(* IEC 61131-3 sources: stformat/handlers/testdata, 60 files *)

(* ---- dut_pragma.golden.iecst ---- *)
{attribute 'qualified_only'}

TYPE S :
	( // Some comment
		A := 10,
		B := 20,
		C := 30,
		D := 40,
		E := 50,
		F := 60,
		G := 70,
		H := 80,
		I := 90,
		J := 100,
		K := 110,
		L := 120,
		M := 130,
		N := 140,
		P := 150
	);
END_TYPE

(* ---- dut_pragma.in.iecst ---- *)
{attribute 'qualified_only'}

TYPE S :
	(  // Some comment
		A := 10, B := 20, C := 30, D := 40, E := 50, F := 60, G := 70, H := 80, I := 90, J := 100, K := 110, L := 120, M := 130, N := 140, P := 150
	);
END_TYPE

(* ---- type_body.golden.st ---- *)
// The value list of a TYPE.
// A TYPE body is a list of values like a call's argument list, so it breaks at the same limit into the same layout.
// The bracket depth is carried from line to line, and text that is not structure must not feed it.

// A body over the limit breaks one member per line.

TYPE EState :
	(
		A := 0,
		B := 1,
		C := 2,
		D := 3,
		E := 4,
		F := 5,
		G := 6,
		H := 7,
		I := 8,
		J := 9,
		K := 10,
		L := 11,
		M := 12,
		N := 13,
		O := 14,
		P := 15
	);
END_TYPE

// One member cannot be split any further, so the line stays long.

TYPE t :
	(
		A := 1000000000000000000000000000000000000000000000000000000000000000000000000000000000000000000000000000000000
	);
END_TYPE

// A parenthesis inside a comment is text, so it does not open a level.
(* note ( unbalanced *)

TYPE FromComment :
	(
		A := 0,
		B := 1,
		C := 2,
		D := 3,
		E := 4,
		F := 5,
		G := 6,
		H := 7,
		I := 8,
		J := 9,
		K := 10,
		L := 11,
		M := 12,
		N := 13,
		O := 14,
		P := 15
	);
END_TYPE

// Same for an ignored region: the count restarts at stformat:on.

TYPE FromRegion :
	// stformat:off
weird ( unbalanced ( ( (
	// stformat:on
	(
		A := 0,
		B := 1,
		C := 2,
		D := 3,
		E := 4,
		F := 5,
		G := 6,
		H := 7,
		I := 8,
		J := 9,
		K := 10,
		L := 11,
		M := 12,
		N := 13,
		O := 14,
		P := 15
	);
END_TYPE

(* ---- type_body.in.st ---- *)
// The value list of a TYPE.
// A TYPE body is a list of values like a call's argument list, so it breaks at the same limit into the same layout.
// The bracket depth is carried from line to line, and text that is not structure must not feed it.

// A body over the limit breaks one member per line.
TYPE EState :
(A := 0, B := 1, C := 2, D := 3, E := 4, F := 5, G := 6, H := 7, I := 8, J := 9, K := 10, L := 11, M := 12, N := 13, O := 14, P := 15);
END_TYPE

// One member cannot be split any further, so the line stays long.
TYPE t :
(A := 1000000000000000000000000000000000000000000000000000000000000000000000000000000000000000000000000000000000);
END_TYPE

// A parenthesis inside a comment is text, so it does not open a level.
(* note ( unbalanced *)
TYPE FromComment :
(A := 0, B := 1, C := 2, D := 3, E := 4, F := 5, G := 6, H := 7, I := 8, J := 9, K := 10, L := 11, M := 12, N := 13, O := 14, P := 15);
END_TYPE

// Same for an ignored region: the count restarts at stformat:on.
TYPE FromRegion :
// stformat:off
weird ( unbalanced ( ( (
// stformat:on
(A := 0, B := 1, C := 2, D := 3, E := 4, F := 5, G := 6, H := 7, I := 8, J := 9, K := 10, L := 11, M := 12, N := 13, O := 14, P := 15);
END_TYPE

(* ---- types.golden.st ---- *)
TYPE point :
	STRUCT
		x : INT;
		y : INT;
	END_STRUCT

	union32 : UNION
		a : INT;
		b : DWORD;
		c : REAL;
	END_UNION

	matrix : ARRAY[1..3, 1..3] OF REAL;
	point_arr : ARRAY[1..4] OF point;
END_TYPE

(* ---- types.in.st ---- *)
type
point:
struct
x: int;
y: int;
end_struct
union32:
union
a: int;
b: dword;
c: real;
end_union
matrix: array[1..3,1..3] of real;
point_arr: array[1..4] of point;
end_type

(* ---- comments.golden.st ---- *)
PROGRAM p
VAR
	x : INT; // the counter
END_VAR

x := 1; // set x
(* block
comment *)
z := 2;
IF x THEN
	y := x; // branch
END_IF // done
(* note *)
z := 3;
END_PROGRAM

// A comment standing on its own line inside a condition.
// The tokens around it ask for no line break, so a second pass used to glue it to the line above.

PROGRAM p
IF a
// both must be set
AND b THEN
	c := 1;
END_IF
END_PROGRAM

// A trailing comment on a condition that has to wrap moves to the THEN line.

PROGRAM p
IF flagOperationalReady
	AND flagMaintenanceOverride
	AND flagEmergencyStopActive
	AND flagPowerAvailable
	AND flagGateClosed
	AND flagInterlockEngaged
	AND flagSequenceRunning
	AND flagAbortRequested
	AND flagResetPermitted
	AND flagCycleComplete
	AND flagAutoModeSelected
THEN // all flags
	x := TRUE;
END_IF
END_PROGRAM

FUNCTION_BLOCK fb EXTENDS base
// built by the comment test
VAR
	y : INT;
END_VAR

y := 1;
END_FUNCTION_BLOCK

// a type with the comment on the line that opens its body

TYPE states :
	(
		// the state names
		a := 0,
		b := 1
	);
END_TYPE

FUNCTION_BLOCK child PUBLIC EXTENDS base
// inherits from base
VAR
	w : INT;
END_VAR
END_FUNCTION_BLOCK
(*****************)
//////////
///doc comment
// x := 1; commented-out code keeps its case
//   indented text keeps its indentation

(* ---- comments.in.st ---- *)
program p
VAR
x:int; //the counter
END_VAR
x:=1; //set x
(* block
comment *)
z:=2;
if x then
    y:=x; //branch
end_if //done
(* note *) z := 3;
end_program

// A comment standing on its own line inside a condition.
// The tokens around it ask for no line break, so a second pass used to glue it to the line above.
program p
IF a
// both must be set
AND b THEN c := 1; END_IF
end_program

// A trailing comment on a condition that has to wrap moves to the THEN line.
program p
IF flagOperationalReady AND flagMaintenanceOverride AND flagEmergencyStopActive AND flagPowerAvailable AND flagGateClosed AND flagInterlockEngaged AND flagSequenceRunning AND flagAbortRequested AND flagResetPermitted AND flagCycleComplete AND flagAutoModeSelected THEN // all flags
    x := TRUE;
END_IF
end_program

function_block fb extends base
// built by the comment test
var
    y:int;
end_var
y:=1;
end_function_block

// a type with the comment on the line that opens its body
type states :
(
// the state names
a:=0,
b:=1
);
end_type

function_block child public extends base
// inherits from base
var
    w:int;
end_var
end_function_block
(*****************)
//////////
///doc comment
//x := 1; commented-out code keeps its case
//   indented text keeps its indentation

(* ---- constructs.golden.st ---- *)
// Namespaces, configurations, property accessors and SFC, whose openers are
// recognised only where their closing keyword follows.

NAMESPACE Motion

FUNCTION F_A : INT
F_A := 1;
END_FUNCTION

FUNCTION F_B : INT
F_B := 2;
END_FUNCTION
END_NAMESPACE

CONFIGURATION Cell
	VAR_GLOBAL
		bRun : BOOL;
	END_VAR

	RESOURCE Cpu ON PLC
		TASK Fast(INTERVAL := T#10MS, PRIORITY := 1);
		PROGRAM Main WITH Fast : P_Main;
	END_RESOURCE
END_CONFIGURATION

FUNCTION_BLOCK FB_Prop
PROPERTY Value : INT
GET
Value := nValue;
END_GET
SET
nValue := Value;
END_SET
END_PROPERTY
END_FUNCTION_BLOCK

PROGRAM Chart
INITIAL_STEP Idle:
	Reset(N);
END_STEP

STEP Run:
	Drive(N);
END_STEP

TRANSITION FROM Idle TO Run := bStart;
END_TRANSITION
END_PROGRAM

// The same words used as names stay names.

PROGRAM Names
VAR
	Step, Set, Get : INT;
END_VAR

Step := Step + 1;
Set := Get;
fb.Set(1);
IF Step > 3 THEN
	Step := 0;
END_IF
END_PROGRAM

// An opener right after a POU header, with no VAR block between.

PROGRAM Direct
STEP Run:
	DriveTheAxisToPosition(Position := fTargetPositionInMillimetres, Velocity := fVelocityLimit, Acceleration := fAcc);
END_STEP
END_PROGRAM

(* ---- constructs.in.st ---- *)
// Namespaces, configurations, property accessors and SFC, whose openers are
// recognised only where their closing keyword follows.
NAMESPACE Motion
FUNCTION F_A : INT
F_A := 1;
END_FUNCTION
FUNCTION F_B : INT
F_B := 2;
END_FUNCTION
END_NAMESPACE

CONFIGURATION Cell
VAR_GLOBAL bRun : BOOL; END_VAR
RESOURCE Cpu ON PLC
TASK Fast(INTERVAL := T#10MS, PRIORITY := 1);
PROGRAM Main WITH Fast : P_Main;
END_RESOURCE
END_CONFIGURATION

FUNCTION_BLOCK FB_Prop
PROPERTY Value : INT
GET
Value := nValue;
END_GET
SET
nValue := Value;
END_SET
END_PROPERTY
END_FUNCTION_BLOCK

PROGRAM Chart
INITIAL_STEP Idle: Reset(N);
END_STEP
STEP Run: Drive(N);
END_STEP
TRANSITION FROM Idle TO Run := bStart;
END_TRANSITION
END_PROGRAM

// The same words used as names stay names.
PROGRAM Names
VAR Step, Set, Get : INT; END_VAR
Step := Step + 1;
Set := Get;
fb.Set(1);
IF Step > 3 THEN Step := 0; END_IF
END_PROGRAM

// An opener right after a POU header, with no VAR block between.
PROGRAM Direct
STEP Run:
DriveTheAxisToPosition(Position := fTargetPositionInMillimetres, Velocity := fVelocityLimit, Acceleration := fAcc);
END_STEP
END_PROGRAM

(* ---- functions.golden.st ---- *)
FUNCTION max2 : INT
max2 := a;
END_FUNCTION

FUNCTION_BLOCK motor
VAR_INPUT
	cmd : BOOL;
	speed : REAL;
END_VAR

METHOD Execute : BOOL
VAR
	result : BOOL;
END_VAR

result := cmd;
END_METHOD
ACTION do_it
speed := 10.0;
END_ACTION
END_FUNCTION_BLOCK

FUNCTION combine : INT
combine := max2(1, 2);
END_FUNCTION

(* ---- functions.in.st ---- *)
function max2: int
max2:=a;
end_function
function_block motor
var_input
cmd: bool;
speed: real;
end_var
method Execute: bool
var
result: bool;
end_var
result:=cmd;
end_method
action do_it
speed:=10.0;
end_action
end_function_block
function combine: int
combine:=max2(1,2);
end_function

(* ---- headers.golden.st ---- *)
// POU and member headers: modifiers, return types and inheritance lists.

FUNCTION F_Ptr : POINTER TO INT
VAR_INPUT
	a : INT;
END_VAR

F_Ptr := ADR(a);
END_FUNCTION

FUNCTION F_Arr : ARRAY[0..1, 1..2] OF INT
END_FUNCTION

FUNCTION F_Str : STRING(80)
END_FUNCTION

FUNCTION F_Ns : Lib.ST_Data
END_FUNCTION

FUNCTION_BLOCK PUBLIC ABSTRACT FB_X EXTENDS FB_Base IMPLEMENTS I_A, Lib.I_B
VAR
END_VAR

METHOD PUBLIC ABSTRACT M : REFERENCE TO INT
VAR_INPUT
	x : INT;
END_VAR
END_METHOD

METHOD FINAL PROTECTED M2 : BOOL
END_METHOD

PROPERTY PUBLIC P : POINTER TO FB_X
END_PROPERTY
END_FUNCTION_BLOCK

INTERFACE I_A EXTENDS I_Base, I_Other
METHOD M : BOOL
END_METHOD
END_INTERFACE

FUNCTION_BLOCK FB_G
VAR_GENERIC CONSTANT
	N : UDINT := 10;
END_VAR
END_FUNCTION_BLOCK

(* ---- headers.in.st ---- *)
// POU and member headers: modifiers, return types and inheritance lists.
FUNCTION F_Ptr : POINTER TO INT
VAR_INPUT a:INT; END_VAR
F_Ptr := ADR(a);
END_FUNCTION

function F_Arr : array[0..1, 1..2] of int
END_FUNCTION

FUNCTION F_Str : STRING(80)
END_FUNCTION

FUNCTION F_Ns : Lib.ST_Data
END_FUNCTION

function_block public abstract FB_X extends FB_Base implements I_A, Lib.I_B
VAR END_VAR

METHOD public abstract M : reference to INT
VAR_INPUT x : INT; END_VAR
END_METHOD

METHOD final protected M2 : BOOL
END_METHOD

PROPERTY PUBLIC P : POINTER TO FB_X
END_PROPERTY
END_FUNCTION_BLOCK

INTERFACE I_A EXTENDS I_Base, I_Other
METHOD M : BOOL
END_METHOD
END_INTERFACE

FUNCTION_BLOCK FB_G
VAR_GENERIC CONSTANT
N : UDINT := 10;
END_VAR
END_FUNCTION_BLOCK

(* ---- oostuff.golden.st ---- *)
CLASS my_class EXTENDS base
VAR
	x : INT;
END_VAR

METHOD PUBLIC compute : INT
compute := x * 2;
END_METHOD
METHOD PROTECTED helper : INT
helper := THIS.x + SUPER.get();
END_METHOD
METHOD ABSTRACT enforce
END_METHOD
METHOD FINAL lockit
register := 1;
END_METHOD
PROPERTY PRIVATE value : INT
END_PROPERTY
END_CLASS

INTERFACE my_interface
METHOD PUBLIC cycle : INT
END_METHOD
METHOD PROTECTED semi : INT
END_METHOD
END_INTERFACE

FUNCTION_BLOCK axis IMPLEMENTS i_motion
VAR
	pos : INT;
END_VAR

METHOD PUBLIC move : INT
move := pos;
END_METHOD
END_FUNCTION_BLOCK

(* ---- oostuff.in.st ---- *)
class my_class extends base
var
x: int;
end_var
method public compute: int
compute:=x*2;
end_method
method protected helper: int
helper:=this.x + super.get();
end_method
method abstract enforce
end_method
method final lockit
register:=1;
end_method
property private value: int
end_property
end_class
interface my_interface
method public cycle: int
end_method
method protected semi: int
end_method
end_interface
function_block axis implements i_motion
var
pos: int;
end_var
method public move: int
move:=pos;
end_method
end_function_block

(* ---- addresses.golden.st ---- *)
PROGRAM p
VAR
	inBit : BOOL AT %i*;
	outBit : BOOL AT %q*;
	inByte : BYTE AT %ib3;
	inWord : WORD AT %IW50;
	outBit2 : BOOL AT %Q0.0;
	memWord : WORD AT %MW100;
	memByte : BYTE AT %MB128;
	memDword : DWORD AT %MD1000;
	memBit : BOOL AT %M0.3;
END_VAR
END_PROGRAM

(* ---- addresses.in.st ---- *)
program p
var
inBit: bool at %i*;
outBit: bool at %q*;
inByte: byte at %ib3;
inWord: word at %IW50;
outBit2: bool at %Q0.0;
memWord: word at %MW100;
memByte: byte at %MB128;
memDword: dword at %MD1000;
memBit: bool at %M0.3;
end_var
end_program

(* ---- bindings.golden.st ---- *)
PROGRAM p
VAR
	setOut : BOOL;
	resetOut : BOOL;
	bitUp : BOOL;
	bitDown : BOOL;
	pSrc : POINTER TO INT;
	pDst : POINTER TO INT;
	pref : REFERENCE TO INT;
	refTo : REF_TO INT;
	pInst : POINTER TO INT;
	pTmp : POINTER TO INT;
	valid : BOOL;
	rAxis : REAL;
	fb : fb_axis;
END_VAR

setOut s= bitUp;
resetOut r= bitDown;
pDst ref= pSrc;
pDst^ := 1;
pref^ := 2;
refTo := fb;
pInst := __NEW(pTmp);
__DELETE(pInst);
valid := __ISVALIDREF(pref);
rAxis := fb.mv(velocity := 100.0);
END_PROGRAM

(* ---- bindings.in.st ---- *)
program p
var
setOut: bool;
resetOut: bool;
bitUp: bool;
bitDown: bool;
pSrc: pointer to int;
pDst: pointer to int;
pref: reference to int;
refTo: ref_to int;
pInst: pointer to int;
pTmp: pointer to int;
valid: bool;
rAxis: real;
fb: fb_axis;
end_var
setOut s= bitUp;
resetOut r= bitDown;
pDst ref= pSrc;
pDst^ := 1;
pref^ := 2;
refTo := fb;
pInst := __NEW(pTmp);
__DELETE(pInst);
valid := __ISVALIDREF(pref);
rAxis := fb.mv(velocity := 100.0);
end_program

(* ---- bom.golden.st ---- *)
// A UTF-8 byte order mark is kept.

PROGRAM bom
x := 1;
END_PROGRAM

(* ---- bom.in.st ---- *)
// A UTF-8 byte order mark is kept.
PROGRAM bom
x:=1;
END_PROGRAM

(* ---- control_flow.golden.st ---- *)
PROGRAM p
VAR
	x : BOOL;
	y : INT;
END_VAR

IF x THEN
	x := TRUE;
ELSIF y > 3 THEN
	y := y + 1;
ELSE
	y := 0;
END_IF

FOR i := 1 TO 10 BY 2 DO
	IF y > 5 THEN
		EXIT;
	END_IF

	i := i + 1;
END_FOR

WHILE x DO
	x := FALSE;
END_WHILE

REPEAT
	y := y - 1;
UNTIL y = 0
END_REPEAT

CASE i OF
	1:
		x := TRUE;

	2, 3:
		y := 5;

	4:
		IF x THEN
			x := TRUE;
		END_IF

	5:
		y := 7;
	ELSE
		y := 0;
END_CASE
END_PROGRAM

(* ---- control_flow.in.st ---- *)
program p
var
x: bool;
y: int;
end_var
if x then
x:=true;
elsif y>3 then
y:=y+1;
else
y:=0;
end_if
for i:=1 to 10 by 2 do
if y>5 then
exit;
end_if
i:=i+1;
end_for
while x do
x:=false;
end_while
repeat
y:=y-1;
until y=0 end_repeat
case i of
1: x:=true;
2,3: y:=5;
4:
if x then
x:=true;
end_if 5: y:=7;
else y:=0;
end_case
end_program

(* ---- directives.golden.st ---- *)
PROGRAM Sections
VAR
	a : INT;
END_VAR

// stformat:off
VAR
	ugly    :   INT;
END_VAR
// stformat:on

a := 1; // stformat:off
   b   :=   2;
// stformat:on

(* stformat:off *)
	untouched   :=   1;
(* stformat:on *)

// STFORMAT: OFF
   another    :=   2;
// stformat : on

// stformat:ignore is only a directive in the leading comment block, so here it
// is an ordinary comment.
b := 4; // stformat:ignore
c := 5;

IF a > 0 THEN
	aLongFunctionName(
		firstArgument := aValueWithALongName,
		secondArgument := anotherValueWithALongName,
		thirdArgument := yetAnotherValue
	); // an explanation of the call
END_IF
END_PROGRAM

(* ---- directives.in.st ---- *)
PROGRAM Sections
VAR
	a : INT;
END_VAR

// stformat:off
VAR
	ugly    :   INT;
END_VAR
// stformat:on

a := 1; // stformat:off
   b   :=   2;
// stformat:on

(* stformat:off *)
	untouched   :=   1;
(* stformat:on *)

// STFORMAT: OFF
   another    :=   2;
// stformat : on

// stformat:ignore is only a directive in the leading comment block, so here it
// is an ordinary comment.
b := 4; // stformat:ignore
c := 5;

IF a > 0 THEN
	aLongFunctionName(firstArgument := aValueWithALongName, secondArgument := anotherValueWithALongName, thirdArgument := yetAnotherValue); // an explanation of the call
END_IF
END_PROGRAM

(* ---- expressions.golden.st ---- *)
PROGRAM p
x := (a AND_THEN b) OR_ELSE (c XOR d);
y := NOT(a AND b);
z := a MOD 7;
w := x ** 2;
q := (len > 0) AND (val <> 0);
cmp := (p^ <> meta.q) OR (r <= 5.0);
END_PROGRAM

(* ---- expressions.in.st ---- *)
program p
x := (a and_then b) or_else (c xor d);
y := not (a and b);
z := a mod 7;
w := x ** 2;
q := (len > 0) and (val <> 0);
cmp := (p^ <> meta.q) or (r <= 5.0);
end_program

(* ---- ignore.golden.st ---- *)
// stformat:ignore
PROGRAM Untouched
    x:=1;
IF   x>0   THEN
	y:=2;
END_IF
END_PROGRAM

(* ---- ignore.in.st ---- *)
// stformat:ignore
PROGRAM Untouched
    x:=1;
IF   x>0   THEN
	y:=2;
END_IF
END_PROGRAM

(* ---- illegal.golden.st ---- *)
// Characters that are not ST are kept, with the spacing they had.

PROGRAM illegal
x := y ? 1;
x := y?1;
a := b&c;
Drehzahl_Ä := Größe;
END_PROGRAM

(* ---- illegal.in.st ---- *)
// Characters that are not ST are kept, with the spacing they had.
PROGRAM illegal
x:=y ? 1;
x:=y?1;
a:=b&c;
Drehzahl_Ä:=Größe;
END_PROGRAM

(* ---- line_breaks.golden.st ---- *)
// Line breaks in the source are kept where they mean something, and dropped everywhere else.
// A break after an opening bracket, around a comma or before a closing bracket keeps that list
// broken open, one item per line. A break before or after an operator keeps that chain broken.

// The list is broken in the source, so it stays broken although it fits.

PROGRAM keptList
result := Combine(
	first := 1,
	second := 2
);
END_PROGRAM

// A break after a comma is enough.

PROGRAM keptListAtComma
result := Combine(
	first := 1,
	second := 2
);
END_PROGRAM

// The chain is broken in the source, so every operator of it starts a line.

PROGRAM keptChain
total := a
	+ b
	+ c;
END_PROGRAM

// The break can also come before the operator.

PROGRAM keptChainBefore
ready := sensorOne
	AND sensorTwo
	AND sensorThree;
END_PROGRAM

// A broken condition is laid out in full.

PROGRAM keptCondition
IF a
	OR b
THEN
	x := 1;
END_IF
END_PROGRAM

// Breaks anywhere else are dropped: after the assignment, between a name and its bracket,
// and inside a list that is not broken at one of its own break points.

PROGRAM dropped
x := 5;
y := F(first := 1, second := 2);
z := Compute(a := 1);
END_PROGRAM

// A broken enum stays broken; one written on a line stays on it.

TYPE E_Broken :
	(
		Idle := 0,
		Running := 1
	);
END_TYPE

TYPE E_Inline :
	(
		Idle := 0,
		Running := 1
	);
END_TYPE

(* ---- line_breaks.in.st ---- *)
// Line breaks in the source are kept where they mean something, and dropped everywhere else.
// A break after an opening bracket, around a comma or before a closing bracket keeps that list
// broken open, one item per line. A break before or after an operator keeps that chain broken.

// The list is broken in the source, so it stays broken although it fits.
PROGRAM keptList
result := Combine(
    first := 1, second := 2);
END_PROGRAM

// A break after a comma is enough.
PROGRAM keptListAtComma
result := Combine(first := 1,
    second := 2);
END_PROGRAM

// The chain is broken in the source, so every operator of it starts a line.
PROGRAM keptChain
total := a +
    b + c;
END_PROGRAM

// The break can also come before the operator.
PROGRAM keptChainBefore
ready := sensorOne
    AND sensorTwo AND sensorThree;
END_PROGRAM

// A broken condition is laid out in full.
PROGRAM keptCondition
IF a
    OR b THEN
    x := 1;
END_IF
END_PROGRAM

// Breaks anywhere else are dropped: after the assignment, between a name and its bracket,
// and inside a list that is not broken at one of its own break points.
PROGRAM dropped
x :=
    5;
y := F(first :=
    1, second := 2);
z := Compute
    (a := 1);
END_PROGRAM

// A broken enum stays broken; one written on a line stays on it.
TYPE E_Broken :
(
    Idle := 0,
    Running := 1
);
END_TYPE

TYPE E_Inline :
(Idle := 0, Running := 1);
END_TYPE

(* ---- literal_spans.golden.st ---- *)
// A literal's text must stop where the literal stops.
// A duration that runs into the code after it swallows that code, and a string spanning lines gets a line break put inside quoted text.

// The duration payload stops at the unit. "T#0MS THEN" read as one token loses the rest of the line.

PROGRAM durationThen
IF i_risingDebounceTime <> T#0MS THEN
	m_risingDebounceTimer(IN := m_state, PT := i_risingDebounceTime);
	IF m_risingDebounceTimer.Q THEN
		updateDebounceState := TRUE;
	END_IF
END_IF

IF x > T#0S THEN
	y := z;
END_IF
END_PROGRAM

// The same, with the assignment and the call after the literal.

PROGRAM durationThenMore
IF t^.p > T#0MS THEN
	p := t^.p;
END_IF

IF r <> T#0S THEN
	a := b := r;
END_IF

IF timer.Q OR d = T#0MS THEN
	c := s;
END_IF

IF ts.e > T#0MS THEN
	x := ts.a + ts.b + ts.c;
END_IF

IF ts.e > T#0MS THEN
	calc(IN := TRUE);
END_IF
END_PROGRAM

// A duration with spaced components is one literal, so the blank inside it is kept.

PROGRAM durationSpaced
a := T#1h 30m 20s;
b := LT#2d 12h;
c := TIME#500ms;
d := T#0MS;
END_PROGRAM

// A string spanning lines is one token, so the comma on the next line is content.

PROGRAM stringSpanningLines
log(
	a := 1,
	fmt := 'first,
second',
	b := 2
);
END_PROGRAM

(* ---- literal_spans.in.st ---- *)
// A literal's text must stop where the literal stops.
// A duration that runs into the code after it swallows that code, and a string spanning lines gets a line break put inside quoted text.

// The duration payload stops at the unit. "T#0MS THEN" read as one token loses the rest of the line.
PROGRAM durationThen
IF i_risingDebounceTime <> T#0MS THEN m_risingDebounceTimer(IN := m_state, PT := i_risingDebounceTime);
IF m_risingDebounceTimer.Q THEN updateDebounceState := TRUE; END_IF END_IF
IF x > T#0S THEN y := z;
END_IF
END_PROGRAM

// The same, with the assignment and the call after the literal.
PROGRAM durationThenMore
IF t^.p > T#0MS THEN p := t^.p; END_IF
IF r <> T#0S THEN a := b := r; END_IF
IF timer.Q OR d = T#0MS  THEN c := s; END_IF
IF ts.e > T#0MS THEN x := ts.a + ts.b + ts.c; END_IF
IF ts.e > T#0MS THEN calc(IN := TRUE);
END_IF
END_PROGRAM

// A duration with spaced components is one literal, so the blank inside it is kept.
PROGRAM durationSpaced
a:=T#1h 30m 20s;
b:=LT#2d 12h;
c:=TIME#500ms;
d:=T#0MS;
END_PROGRAM

// A string spanning lines is one token, so the comma on the next line is content.
PROGRAM stringSpanningLines
log(
a := 1,
fmt := 'first,
second',
b := 2
);
END_PROGRAM

(* ---- literals.golden.st ---- *)
PROGRAM p
VAR
	hexVal : DWORD := 16#FF;
	binVal : BYTE := 2#1011;
	octVal : BYTE := 8#77;
	mask : DWORD := 16#FFFFFFFF;
	intTyped : DINT := DINT#-32768;
	wordTyped : WORD := WORD#16#ABCD;
	realTyped : REAL := REAL#1.5;
	boolTyped : BOOL := BOOL#TRUE;
	expVal : REAL := 1.5e3;
	negExp : LREAL := 1.5E-3;
	dur1 : TIME := T#1H 30M 20S 500MS;
	dur2 : TIME := TIME#5S;
	dur3 : LTIME := LTIME#100NS;
	todVal : TOD := TOD#12:30:45.5;
	dateVal : DATE := DATE#2024-06-15;
	dtVal : DT := DT#2024-06-15-12:30:45;
	ldtVal : LDT := LDT#2024-06-15-12:30:45.123;
	str1 : STRING := 'plain';
	str2 : WSTRING := "line1$R$Nline2";
	str3 : STRING := STRING#'typed';
	str4 : STRING := STRING#"typed";
	str5 : WSTRING := WSTRING#'typed';
	str6 : WSTRING := WSTRING#"typed";
	ch1 : CHAR := CHAR#'a';
	ch2 : CHAR := CHAR#"b";
	wch1 : WCHAR := WCHAR#"ab";
	sep : LREAL := 1_0E1_0;
	expSep : LREAL := 1.5E1_0;
	negDur : LTIME := LTIME#-5s;
END_VAR
END_PROGRAM

(* ---- literals.in.st ---- *)
program p
var
hexVal: dword := 16#FF;
binVal: byte := 2#1011;
octVal: byte := 8#77;
mask: dword := 16#FFFFFFFF;
intTyped: dint := DINT#-32768;
wordTyped: word := WORD#16#ABCD;
realTyped: real := REAL#1.5;
boolTyped: bool := BOOL#TRUE;
expVal: real := 1.5e3;
negExp: lreal := 1.5E-3;
dur1: time := T#1H 30M 20S 500MS;
dur2: time := TIME#5S;
dur3: ltime := LTIME#100NS;
todVal: tod := TOD#12:30:45.5;
dateVal: date := DATE#2024-06-15;
dtVal: dt := DT#2024-06-15-12:30:45;
ldtVal: ldt := LDT#2024-06-15-12:30:45.123;
str1: string := 'plain';
str2: wstring := "line1$R$Nline2";
str3: string := STRING#'typed';
str4: string := STRING#"typed";
str5: wstring := WSTRING#'typed';
str6: wstring := WSTRING#"typed";
ch1: char := CHAR#'a';
ch2: char := CHAR#"b";
wch1: wchar := WCHAR#"ab";
sep: lreal := 1_0E1_0;
expSep: lreal := 1.5E1_0;
negDur: ltime := LTIME#-5s;
end_var
end_program

(* ---- long_call.golden.st ---- *)
PROGRAM p
cmd.FB_Build(
	rDoExtending := rDoExtending,
	rDoRetracting := rDoRetracting,
	rDiAtExtendedPosition := rDiAtExtendedPosition,
	rDiAtRetractedPosition := rDiAtRetractedPosition,
	commandTimeout := T#5S,
	driveEnable := TRUE,
	speedFactor := 1.0
);
cmd.FB_Build(a := 1, b := 2);
END_PROGRAM

(* ---- long_call.in.st ---- *)
program p
cmd.FB_Build(rDoExtending:=rDoExtending, rDoRetracting:=rDoRetracting, rDiAtExtendedPosition:=rDiAtExtendedPosition, rDiAtRetractedPosition:=rDiAtRetractedPosition, commandTimeout:=T#5S, driveEnable:=TRUE, speedFactor:=1.0);
cmd.FB_Build(a:=1, b:=2);
end_program

(* ---- members.golden.st ---- *)
// Members and enum values spelled like keywords stay identifiers.

PROGRAM members
stData.Type := 1;
x := msg.Final;
y := a.Exit;
b := c.Var;
IF fb.Method() THEN
	fb.Action();
END_IF

e := E_Kind.Interface;
t := stLog.Time;
END_PROGRAM

(* ---- members.in.st ---- *)
// Members and enum values spelled like keywords stay identifiers.
PROGRAM members
stData.Type:=1;
x:=msg.Final;
y:=a.Exit;
b:=c.Var;
IF fb.Method() THEN fb.Action(); END_IF
e:=E_Kind.Interface;
t:=stLog.Time;
END_PROGRAM

(* ---- program_shape.golden.st ---- *)
// What the formatter does to a whole file rather than to a line.
// Blank lines between POUs, after a declaration block and after a block end are its own decisions.

// A POU that does nothing still comes back with a trailing newline.

PROGRAM Untouched
END_PROGRAM

PROGRAM p
x := 1;
END_PROGRAM

// Two POUs in one file are separated by a blank line.

FUNCTION f
END_FUNCTION

FUNCTION g
END_FUNCTION

// A declaration block is separated from the code that follows it.

PROGRAM decl
VAR
	x : BOOL;
END_VAR

x := 1;
END_PROGRAM

// A statement after END_IF starts a new paragraph.

PROGRAM afterEndIf
IF x THEN
	x := TRUE;
END_IF

y := 1;
END_PROGRAM

// The same for a block that ends inside another one.

PROGRAM nestedBlockEnd
FOR i := 1 TO 10 DO
	IF x THEN
		EXIT;
	END_IF

	RETURN;
END_FOR
END_PROGRAM

// An empty program is left alone apart from the trailing newline.

PROGRAM P
END_PROGRAM

(* ---- program_shape.in.st ---- *)
// What the formatter does to a whole file rather than to a line.
// Blank lines between POUs, after a declaration block and after a block end are its own decisions.

// A POU that does nothing still comes back with a trailing newline.
PROGRAM Untouched
END_PROGRAM
PROGRAM p
x:=1;
END_PROGRAM

// Two POUs in one file are separated by a blank line.
FUNCTION f
END_FUNCTION
FUNCTION g
END_FUNCTION

// A declaration block is separated from the code that follows it.
PROGRAM decl
VAR
x : BOOL;
END_VAR
x := 1;
END_PROGRAM

// A statement after END_IF starts a new paragraph.
PROGRAM afterEndIf
IF x THEN
    x := TRUE;
END_IF y:=1;
END_PROGRAM

// The same for a block that ends inside another one.
PROGRAM nestedBlockEnd
FOR i:=1 TO 10 DO
    IF x THEN
        EXIT;
    END_IF
    RETURN;
END_FOR
END_PROGRAM

// An empty program is left alone apart from the trailing newline.
PROGRAM P
END_PROGRAM

(* ---- set_reset.golden.st ---- *)
// S=, R= and REF= follow an assignment target; anywhere else s, r and ref are names.

PROGRAM set_reset
bOut S= bIn;
bOut R= bIn;
pData REF= stData;
arr[1] S= TRUE;
IF s = 1 THEN
	x := 1;
END_IF

IF r = 2 AND ref = 3 THEN
	y := s;
END_IF

b := a = s;
fb(s => q, r => p);
END_PROGRAM

(* ---- set_reset.in.st ---- *)
// S=, R= and REF= follow an assignment target; anywhere else s, r and ref are names.
PROGRAM set_reset
bOut S= bIn;
bOut R= bIn;
pData REF= stData;
arr[1] S= TRUE;
IF s=1 THEN x:=1; END_IF
IF r=2 AND ref=3 THEN y:=s; END_IF
b:=a=s;
fb(s=>q, r=>p);
END_PROGRAM

(* ---- unary.golden.st ---- *)
// Signs bind to their operand; binary + and - keep a space on both sides.

PROGRAM unary
x := -1;
y := a * -b;
z := -(a + b);
w := a - -b;
v := 2 ** -1;
u := a - 1;
t := f(-x, +y);
s := arr[-1] + arr[i] - 1;
IF x < -1 OR y >= -2 THEN
	q := -q;
END_IF

CASE n OF
	-1:
		r := -1;
END_CASE

FOR i := -10 TO -1 BY -1 DO
END_FOR
END_PROGRAM

(* ---- unary.in.st ---- *)
// Signs bind to their operand; binary + and - keep a space on both sides.
PROGRAM unary
x:=-1;
y:=a*-b;
z:=-(a+b);
w:=a - -b;
v:=2**-1;
u:=a-1;
t:=f(-x, +y);
s:=arr[-1]+arr[i]-1;
IF x<-1 OR y>=-2 THEN q:=-q; END_IF
CASE n OF
-1: r:=-1;
END_CASE
FOR i:=-10 TO -1 BY -1 DO END_FOR
END_PROGRAM

(* ---- var_blocks.golden.st ---- *)
PROGRAM p
VAR_INST
	fbInner : fb_motor;
END_VAR

VAR_STAT
	callCount : INT;
END_VAR

VAR_EXTERNAL
	shared : INT;
END_VAR

VAR_CONFIG
	inst.address : BOOL AT %i*;
END_VAR

VAR_ACCESS
	nCount : gvl.nCount : DINT READ_WRITE;
	sSecret : gvl.sSecret : STRING READ_ONLY;
END_VAR

VAR_GLOBAL NON_RETAIN
	cfg : INT;
END_VAR

VAR CONSTANT
	kPi : REAL := 3.14159;
END_VAR

VAR PERSISTENT
	bootCount : DINT;
END_VAR
END_PROGRAM

(* ---- var_blocks.in.st ---- *)
program p
var_inst
fbInner: fb_motor;
end_var
var_stat
callCount: int;
end_var
var_external
shared: int;
end_var
var_config
inst.address: bool at %i*;
end_var
var_access
nCount: gvl.nCount: dint read_write;
sSecret: gvl.sSecret: string read_only;
end_var
var_global non_retain
cfg: int;
end_var
var constant
kPi: real := 3.14159;
end_var
var persistent
bootCount: dint;
end_var
end_program

(* ---- variables.golden.st ---- *)
PROGRAM p
VAR_INPUT
	a : BOOL;
	start_position : REAL := 1.0;
	count : INT;
END_VAR

VAR_OUTPUT
	result : STRING(32);
END_VAR

VAR_TEMP
	tempbuf : ARRAY[1..10] OF INT;
END_VAR

VAR_GLOBAL RETAIN
	max_speed : UDINT := 2000;
END_VAR

VAR
	pin_ptr : POINTER TO INT;
	ref_var : REFERENCE TO BOOL;
	mapped : INT AT %mb30;
END_VAR
END_PROGRAM

(* ---- variables.in.st ---- *)
program p
var_input
a: bool;
start_position: real := 1.0;
count: int;
end_var
var_output
result: string(32);
end_var
var_temp
tempbuf: array[1..10] of int;
end_var
var_global retain
max_speed: udint := 2000;
end_var
var
pin_ptr: pointer to int;
ref_var: reference to bool;
mapped: int at %mb30;
end_var
end_program

(* ---- wrap_boundaries.golden.st ---- *)
// What the wrap must not touch.
// The reflow breaks a line at 120 columns, but only when the line is code.
// Each case below is the same rule against a different kind of not-code.

// A long call inside an ignored region. The region is already how its author wants it.

PROGRAM ignored
// stformat:off
averyveryverylongfunction(firstArgument := aValueWithALongName, secondArgument := anotherValueWithALongName, thirdArgument := yetAnotherValue);
// stformat:on
// The rule ends at stformat:on, so the next long line is wrapped normally.
anotherveryverylongfunction(
	firstArgument := aValueWithALongName,
	secondArgument := anotherValueWithALongName,
	thirdArgument := yetAnotherValue
);
END_PROGRAM

// The short line opens the block comment, so the long line after it is comment text.

PROGRAM blockOpen
(* block
veryveryverylongfunction(firstArgument := aValueWithALongName, secondArgument := anotherValueWithALongName, thirdArgument := yetAnotherValue);
*)
cal(a := 1, b := 2);
END_PROGRAM

// The comment opens and closes on the long line itself, so the next line is code again.

PROGRAM blockClosed
(* a long comment that just goes on and on and on and on and on and on and on and on and on *)
veryveryverylongfunction(
	firstArgument := aValueWithALongName,
	secondArgument := anotherValueWithALongName,
	thirdArgument := yetAnotherValue
);
END_PROGRAM

// An opening delimiter inside a string literal is text, not a comment.

PROGRAM delimiterInString
cal(
	a := 1,
	b := '(* not a comment',
	c := 2,
	d := 3,
	e := 4,
	f := 5,
	g := 6,
	h := 7,
	i := 8,
	j := 9,
	k := 10,
	l := 11,
	m := 12,
	n := 13,
	o := 14,
	p := 15
);
END_PROGRAM

// A comma inside a string literal does not separate arguments.

PROGRAM commaInString
Log(id := 1, msgFmtStr := 'one, two', strArg := 'three');
END_PROGRAM

// A string literal that runs over a line break stays one token; the list the source broke open stays broken.

PROGRAM stringSpanningLines
ADSLOGSTR(
	msgCtrlMask := ADSLOG_MSGTYPE_ERROR OR ADSLOG_MSGTYPE_MSGBOX,
	msgFmtStr := 'addChild: To many subUnits,
%s',
	strArg := sArg
);
END_PROGRAM

// Over 120 columns with a literal that runs onto the next line: the call breaks, the literal is left as it is.

PROGRAM callWithMultilineString
cal(
	a := 1,
	b := 2,
	c := 3,
	d := 4,
	e := 5,
	f := 6,
	g := 7,
	h := 8,
	i := 9,
	j := 10,
	k := 11,
	l := 12,
	m := 13,
	fmt := 'first,
second'
);
END_PROGRAM

(* ---- wrap_boundaries.in.st ---- *)
// What the wrap must not touch.
// The reflow breaks a line at 120 columns, but only when the line is code.
// Each case below is the same rule against a different kind of not-code.

// A long call inside an ignored region. The region is already how its author wants it.
PROGRAM ignored
// stformat:off
averyveryverylongfunction(firstArgument := aValueWithALongName, secondArgument := anotherValueWithALongName, thirdArgument := yetAnotherValue);
// stformat:on
// The rule ends at stformat:on, so the next long line is wrapped normally.
anotherveryverylongfunction(firstArgument := aValueWithALongName, secondArgument := anotherValueWithALongName, thirdArgument := yetAnotherValue);
END_PROGRAM

// The short line opens the block comment, so the long line after it is comment text.
PROGRAM blockOpen
(* block
veryveryverylongfunction(firstArgument := aValueWithALongName, secondArgument := anotherValueWithALongName, thirdArgument := yetAnotherValue);
*)
cal(a := 1, b := 2);
END_PROGRAM

// The comment opens and closes on the long line itself, so the next line is code again.
PROGRAM blockClosed
(* a long comment that just goes on and on and on and on and on and on and on and on and on *)
veryveryverylongfunction(firstArgument := aValueWithALongName, secondArgument := anotherValueWithALongName, thirdArgument := yetAnotherValue);
END_PROGRAM

// An opening delimiter inside a string literal is text, not a comment.
PROGRAM delimiterInString
cal(a := 1, b := '(* not a comment', c := 2, d := 3, e := 4, f := 5, g := 6, h := 7, i := 8, j := 9, k := 10, l := 11, m := 12, n := 13, o := 14, p := 15);
END_PROGRAM

// A comma inside a string literal does not separate arguments.
PROGRAM commaInString
Log(id := 1, msgFmtStr := 'one, two', strArg := 'three');
END_PROGRAM

// A string literal that runs over a line break stays one token; the list the source broke open stays broken.
PROGRAM stringSpanningLines
ADSLOGSTR(
msgCtrlMask := ADSLOG_MSGTYPE_ERROR OR ADSLOG_MSGTYPE_MSGBOX,
msgFmtStr := 'addChild: To many subUnits,
%s',
strArg := sArg
);
END_PROGRAM

// Over 120 columns with a literal that runs onto the next line: the call breaks, the literal is left as it is.
PROGRAM callWithMultilineString
cal(a := 1, b := 2, c := 3, d := 4, e := 5, f := 6, g := 7, h := 8, i := 9, j := 10, k := 11, l := 12, m := 13, fmt := 'first,
second');
END_PROGRAM

(* ---- wrap_calls.golden.st ---- *)
PROGRAM WrapCalls
VAR
	result : BOOL;

	// Array literal whose elements are parenthesized constructor calls.
	// The closing ']' must be preserved when the line overflows.
	slots : ARRAY[0..3] OF ST_SlotConfig[
		(key := 'aaa001', description := 'slot for the alpha lane'),
		(key := 'bbb002', description := 'slot for the beta side'),
		(key := 'ccc003', description := 'slot near the gamma unit'),
		(key := 'ddd004', description := 'slot below the delta frame')
	];
END_VAR

// A call that is not the end of the statement: the trailing
// `AND result` must survive long-line wrapping.
createStatusEventList := m_rejectList.addRejectReason(
	status := GVL_FlowStatus.INVALID,
	pEvent := ADR(m_statusUnknown),
	reasonCode := eReasonCode.Unreadable
) AND createStatusEventList;
END_PROGRAM

(* ---- wrap_calls.in.st ---- *)
PROGRAM WrapCalls
VAR
    result : BOOL;

    // Array literal whose elements are parenthesized constructor calls.
    // The closing ']' must be preserved when the line overflows.
    slots : ARRAY[0..3] OF ST_SlotConfig[
        (key := 'aaa001', description := 'slot for the alpha lane'),
        (key := 'bbb002', description := 'slot for the beta side'),
        (key := 'ccc003', description := 'slot near the gamma unit'),
        (key := 'ddd004', description := 'slot below the delta frame')];
END_VAR

// A call that is not the end of the statement: the trailing
// `AND result` must survive long-line wrapping.
createStatusEventList := m_rejectList.addRejectReason(status := GVL_FlowStatus.INVALID, pEvent := ADR(m_statusUnknown), reasonCode := eReasonCode.Unreadable) AND createStatusEventList;
END_PROGRAM

(* ---- wrap_expressions.golden.st ---- *)
// Any expression that does not fit is broken, not only call lists and IF conditions.
// A list is broken open first; an operator chain breaks before each of its operators,
// one level deeper than the line it starts on.

// Long arithmetic breaks at its lowest operators; the products stay whole.

PROGRAM arithmetic
totalEnergyConsumption := motorPowerPhaseOne * operatingHoursPhaseOne
	+ motorPowerPhaseTwo * operatingHoursPhaseTwo
	+ auxiliaryLoad;
END_PROGRAM

// A long assignment whose right side is a single call keeps the call on the first line.

PROGRAM assignment
resultingConfiguration := ConfigurationBuilder(
	sourceMachine := primaryMachineIdentifier,
	targetLine := productionLineIdentifier
);
END_PROGRAM

// Nested calls: each line the layout produces is laid out again, so a long argument breaks too.

PROGRAM nested
outerCall(
	firstArgument := innerCall(
		alphaParameter := alphaValueWithLongName,
		betaParameter := betaValueWithLongName,
		gammaParameter := gammaValue
	),
	second := 2
);
END_PROGRAM

// A call with one argument is not broken open; the call inside it is.

PROGRAM singleArgument
wrapperFunction(innerFunctionWithLongName(
	firstParameter := firstValueWithLongName,
	secondParameter := secondValueWithLongName
));
END_PROGRAM

// A chain with a call on either side breaks at the operator when breaking the call does not make it fit.

PROGRAM chainOfCalls
isWithinTolerance := ABS(measuredPositionOfTheAxis - commandedPositionOfTheAxis) < positionToleranceOfTheAxis
	AND axisIsEnabled;
END_PROGRAM

// A WHILE condition is laid out like an IF condition.

PROGRAM whileLoop
WHILE conveyorIsRunning
	AND NOT emergencyStopPressed
	AND productDetectedAtInfeed
	AND outfeedIsClear
	AND counter < maximumCount
DO
	counter := counter + 1;
END_WHILE
END_PROGRAM

(* ---- wrap_expressions.in.st ---- *)
// Any expression that does not fit is broken, not only call lists and IF conditions.
// A list is broken open first; an operator chain breaks before each of its operators,
// one level deeper than the line it starts on.

// Long arithmetic breaks at its lowest operators; the products stay whole.
PROGRAM arithmetic
totalEnergyConsumption := motorPowerPhaseOne * operatingHoursPhaseOne + motorPowerPhaseTwo * operatingHoursPhaseTwo + auxiliaryLoad;
END_PROGRAM

// A long assignment whose right side is a single call keeps the call on the first line.
PROGRAM assignment
resultingConfiguration := ConfigurationBuilder(sourceMachine := primaryMachineIdentifier, targetLine := productionLineIdentifier);
END_PROGRAM

// Nested calls: each line the layout produces is laid out again, so a long argument breaks too.
PROGRAM nested
outerCall(firstArgument := innerCall(alphaParameter := alphaValueWithLongName, betaParameter := betaValueWithLongName, gammaParameter := gammaValue), second := 2);
END_PROGRAM

// A call with one argument is not broken open; the call inside it is.
PROGRAM singleArgument
wrapperFunction(innerFunctionWithLongName(firstParameter := firstValueWithLongName, secondParameter := secondValueWithLongName));
END_PROGRAM

// A chain with a call on either side breaks at the operator when breaking the call does not make it fit.
PROGRAM chainOfCalls
isWithinTolerance := ABS(measuredPositionOfTheAxis - commandedPositionOfTheAxis) < positionToleranceOfTheAxis AND axisIsEnabled;
END_PROGRAM

// A WHILE condition is laid out like an IF condition.
PROGRAM whileLoop
WHILE conveyorIsRunning AND NOT emergencyStopPressed AND productDetectedAtInfeed AND outfeedIsClear AND counter < maximumCount DO
    counter := counter + 1;
END_WHILE
END_PROGRAM

(* ---- wrap_if.golden.st ---- *)
PROGRAM WrapIf
VAR
	flagOperationalReady : BOOL;
	flagMaintenanceOverride : BOOL;
	flagEmergencyStopActive : BOOL;
	flagPowerAvailable : BOOL;
	flagGateClosed : BOOL;
	flagInterlockEngaged : BOOL;
	flagSequenceRunning : BOOL;
	flagAbortRequested : BOOL;
	flagResetPermitted : BOOL;
	flagCycleComplete : BOOL;
	flagAutoModeSelected : BOOL;
	flagManualModeSelected : BOOL;
	flagRemoteModeSelected : BOOL;
	flagLocalModeSelected : BOOL;
	result : BOOL;
	cmdText : STRING(80);
END_VAR

// Simple long IF: split at top-level AND.
IF flagOperationalReady
	AND flagMaintenanceOverride
	AND flagEmergencyStopActive
	AND flagPowerAvailable
	AND flagGateClosed
	AND flagInterlockEngaged
	AND flagSequenceRunning
	AND flagAbortRequested
	AND flagResetPermitted
	AND flagCycleComplete
	AND flagAutoModeSelected
THEN
	result := TRUE;
END_IF

// Parenthesised combined condition stays together when it fits.
IF (
		flagOperationalReady
		OR flagMaintenanceOverride
	)
	AND flagEmergencyStopActive
	AND flagPowerAvailable
	AND flagGateClosed
	AND flagInterlockEngaged
	AND flagSequenceRunning
THEN
	result := TRUE;
END_IF

// Over-long combined condition is deep-split at its own AND operators.
IF (
		flagOperationalReady
		AND flagMaintenanceOverride
		AND flagEmergencyStopActive
		AND flagPowerAvailable
		AND flagGateClosed
		AND flagInterlockEngaged
		AND flagSequenceRunning
		AND flagAbortRequested
	)
	AND flagResetPermitted
THEN
	result := TRUE;
END_IF

// ELSIF also wraps.
IF flagOperationalReady THEN
	result := FALSE;
ELSIF flagOperationalReady
	AND flagMaintenanceOverride
	AND flagEmergencyStopActive
	AND flagPowerAvailable
	AND flagGateClosed
	AND flagInterlockEngaged
	AND flagSequenceRunning
	AND flagAbortRequested
THEN
	result := TRUE;
END_IF

// Short IF stays inline.
IF flagOperationalReady AND flagMaintenanceOverride THEN
	result := TRUE;
END_IF

// XOR chain wraps the same way.
IF flagOperationalReady
	OR flagMaintenanceOverride
	OR flagEmergencyStopActive
	OR flagPowerAvailable
	OR flagGateClosed
	OR flagInterlockEngaged
THEN
	result := TRUE;
END_IF

// String literal containing THEN/AND is not split.
cmdText := 'FIND THEN AND OR XOR';
IF cmdText = 'FIND THEN AND OR XOR'
	AND flagOperationalReady
	AND flagMaintenanceOverride
	AND flagEmergencyStopActive
	AND flagPowerAvailable
	AND flagGateClosed
THEN
	result := TRUE;
END_IF

// Mixed AND/OR with two short paren groups.
IF (
		flagOperationalReady
		AND flagMaintenanceOverride
	)
	OR (
		flagEmergencyStopActive
		AND flagPowerAvailable
	)
	AND flagGateClosed
	AND flagInterlockEngaged
	AND flagSequenceRunning
	AND flagAbortRequested
THEN
	result := TRUE;
END_IF

// Over-long first paren group deep-splits; second short group stays whole.
IF (
		flagOperationalReady
		AND flagMaintenanceOverride
		AND flagEmergencyStopActive
		AND flagPowerAvailable
		AND flagGateClosed
		AND flagInterlockEngaged
	)
	OR (
		flagAbortRequested
		AND flagResetPermitted
	)
THEN
	result := TRUE;
END_IF

// Both paren groups overlong: deep-split at two indent levels.
IF (
		flagOperationalReady
		AND flagMaintenanceOverride
		AND flagEmergencyStopActive
		AND flagPowerAvailable
		AND flagGateClosed
		AND flagInterlockEngaged
	)
	OR (
		flagSequenceRunning
		AND flagAbortRequested
		AND flagResetPermitted
		AND flagCycleComplete
		AND flagAutoModeSelected
		AND flagManualModeSelected
	)
THEN
	result := TRUE;
END_IF

// Nested parens inside parens: inner AND/OR stays with its group.
IF (
		(
			flagOperationalReady
			OR flagMaintenanceOverride
		)
		AND (
			flagEmergencyStopActive
			OR flagPowerAvailable
		)
	)
	AND flagGateClosed
	AND flagInterlockEngaged
	AND flagSequenceRunning
	AND flagAbortRequested
THEN
	result := TRUE;
END_IF

// Mixed top-level: multiple paren groups separated by OR, with trailing AND chain.
IF (
		flagOperationalReady
		AND flagMaintenanceOverride
	)
	OR (
		flagEmergencyStopActive
		AND flagPowerAvailable
	)
	OR (
		flagGateClosed
		AND flagInterlockEngaged
	)
	AND flagSequenceRunning
	AND flagAbortRequested
	AND flagResetPermitted
	AND flagCycleComplete
THEN
	result := TRUE;
END_IF
END_PROGRAM

(* ---- wrap_if.in.st ---- *)
PROGRAM WrapIf

VAR
    flagOperationalReady    : BOOL;
    flagMaintenanceOverride : BOOL;
    flagEmergencyStopActive : BOOL;
    flagPowerAvailable      : BOOL;
    flagGateClosed          : BOOL;
    flagInterlockEngaged    : BOOL;
    flagSequenceRunning     : BOOL;
    flagAbortRequested      : BOOL;
    flagResetPermitted      : BOOL;
    flagCycleComplete       : BOOL;
    flagAutoModeSelected    : BOOL;
    flagManualModeSelected  : BOOL;
    flagRemoteModeSelected  : BOOL;
    flagLocalModeSelected   : BOOL;
    result                  : BOOL;
    cmdText                 : STRING(80);
END_VAR

// Simple long IF: split at top-level AND.
IF flagOperationalReady AND flagMaintenanceOverride AND flagEmergencyStopActive AND flagPowerAvailable AND flagGateClosed AND flagInterlockEngaged AND flagSequenceRunning AND flagAbortRequested AND flagResetPermitted AND flagCycleComplete AND flagAutoModeSelected THEN
    result := TRUE;
END_IF

// Parenthesised combined condition stays together when it fits.
IF (flagOperationalReady OR flagMaintenanceOverride) AND flagEmergencyStopActive AND flagPowerAvailable AND flagGateClosed AND flagInterlockEngaged AND flagSequenceRunning THEN
    result := TRUE;
END_IF

// Over-long combined condition is deep-split at its own AND operators.
IF (flagOperationalReady AND flagMaintenanceOverride AND flagEmergencyStopActive AND flagPowerAvailable AND flagGateClosed AND flagInterlockEngaged AND flagSequenceRunning AND flagAbortRequested) AND flagResetPermitted THEN
    result := TRUE;
END_IF

// ELSIF also wraps.
IF flagOperationalReady THEN
    result := FALSE;
ELSIF flagOperationalReady AND flagMaintenanceOverride AND flagEmergencyStopActive AND flagPowerAvailable AND flagGateClosed AND flagInterlockEngaged AND flagSequenceRunning AND flagAbortRequested THEN
    result := TRUE;
END_IF

// Short IF stays inline.
IF flagOperationalReady AND flagMaintenanceOverride THEN
    result := TRUE;
END_IF

// XOR chain wraps the same way.
IF flagOperationalReady OR flagMaintenanceOverride OR flagEmergencyStopActive OR flagPowerAvailable OR flagGateClosed OR flagInterlockEngaged THEN
    result := TRUE;
END_IF

// String literal containing THEN/AND is not split.
cmdText := 'FIND THEN AND OR XOR';
IF cmdText = 'FIND THEN AND OR XOR' AND flagOperationalReady AND flagMaintenanceOverride AND flagEmergencyStopActive AND flagPowerAvailable AND flagGateClosed THEN
    result := TRUE;
END_IF

// Mixed AND/OR with two short paren groups.
IF (flagOperationalReady AND flagMaintenanceOverride) OR (flagEmergencyStopActive AND flagPowerAvailable) AND flagGateClosed AND flagInterlockEngaged AND flagSequenceRunning AND flagAbortRequested THEN
    result := TRUE;
END_IF

// Over-long first paren group deep-splits; second short group stays whole.
IF (flagOperationalReady AND flagMaintenanceOverride AND flagEmergencyStopActive AND flagPowerAvailable AND flagGateClosed AND flagInterlockEngaged) OR (flagAbortRequested AND flagResetPermitted) THEN
    result := TRUE;
END_IF

// Both paren groups overlong: deep-split at two indent levels.
IF (flagOperationalReady AND flagMaintenanceOverride AND flagEmergencyStopActive AND flagPowerAvailable AND flagGateClosed AND flagInterlockEngaged) OR (flagSequenceRunning AND flagAbortRequested AND flagResetPermitted AND flagCycleComplete AND flagAutoModeSelected AND flagManualModeSelected) THEN
    result := TRUE;
END_IF

// Nested parens inside parens: inner AND/OR stays with its group.
IF ((flagOperationalReady OR flagMaintenanceOverride) AND (flagEmergencyStopActive OR flagPowerAvailable)) AND flagGateClosed AND flagInterlockEngaged AND flagSequenceRunning AND flagAbortRequested THEN
    result := TRUE;
END_IF

// Mixed top-level: multiple paren groups separated by OR, with trailing AND chain.
IF (flagOperationalReady AND flagMaintenanceOverride) OR (flagEmergencyStopActive AND flagPowerAvailable) OR (flagGateClosed AND flagInterlockEngaged) AND flagSequenceRunning AND flagAbortRequested AND flagResetPermitted AND flagCycleComplete THEN
    result := TRUE;
END_IF

END_PROGRAM
